// TIA Portal V18 export
DATA_BLOCK "MU_Spin_DB"   // DB31
// stored: AutoNumber false, InstanceOfName MU_Spin, InstanceOfType FB
"MU_Spin"
   // VAR_OUTPUT
   //    FlowFwdmAOut : Real;
   //    TorqmAOut : Real;
   //    FwdEnableP1 : Bool;
   //    FwdEnableP2 : Bool;
   //    TorqEn : Bool;
   // END_VAR
   // VAR
   //    LinkExtSw_Last : Bool;
   //    LinkRetSw_Last : Bool;
   //    MUSpinComplete : Bool;
   // END_VAR
BEGIN
END_DATA_BLOCK
